{attribute 'GeneratedUsingTerminal: EK1122-0000-0018'}
{attribute addProperty BoxType "EK1122-0000-0018"}
{attribute addProperty Id "RP30_VI_AES_D_BC_ECAT_xAES_A3B0707168RP30_SAFETY_Flexi_Soft_EtherCAT_GatewayFlexi_Soft_EtherCAT_Gateway_DE394EDD5RP30_AB0_EPP1322_0001EPP1322_1FC0878B2RP30_AB1_EPP1008_0001EPP1008_78E8D3DD12RP30_AB2_EPP1008_0001EPP1008_78E8D3DD12RP30_AB3_EPP1008_0001EPP1008_78E8D3DD12RP30_AB4_EPP1008_0001EPP1008_78E8D3DD12"}
{attribute addProperty CRC "3284966580"}
{attribute addProperty Size "123"}
{attribute addProperty Name "RP30_A2 (EK1122)"}
TYPE RP30_A2_EK1122_C3CC9CB4 EXTENDS EK1122_1FC0878B :
STRUCT
    {attribute addProperty Name "RP30-VI (AES-D-BC-ECAT)"}
    {attribute addProperty PreviousPort "RP30_A2 (EK1122) : D"}
    {attribute addProperty SyncUnit "P30"}
    RP30_VI_AES_D_BC_ECAT_x : AES_A3B07071;
    {attribute addProperty Name "RP30-SAFETY (Flexi Soft EtherCAT Gateway)"}
    {attribute addProperty PreviousPort "RP30_A2 (EK1122) : B"}
    {attribute addProperty SyncUnit "P30"}
    RP30_SAFETY_Flexi_Soft_EtherCAT_Gateway : Flexi_Soft_EtherCAT_Gateway_DE394EDD;
    {attribute addProperty Name "RP30-AB0 (EPP1322-0001)"}
    {attribute addProperty PreviousPort "RP30-SAFETY (Flexi Soft EtherCAT Gateway) : B"}
    {attribute addProperty SyncUnit "default"}
    RP30_AB0_EPP1322_0001 : EPP1322_1FC0878B;
    {attribute addProperty Name "RP30-AB1 (EPP1008-0001)"}
    {attribute addProperty PreviousPort "RP30-AB0 (EPP1322-0001) : C"}
    {attribute addProperty SyncUnit "P30"}
    RP30_AB1_EPP1008_0001 : EPP1008_78E8D3DD;
    {attribute addProperty Name "RP30-AB2 (EPP1008-0001)"}
    {attribute addProperty PreviousPort "RP30-AB1 (EPP1008-0001) : B"}
    {attribute addProperty SyncUnit "P30"}
    RP30_AB2_EPP1008_0001 : EPP1008_78E8D3DD;
    {attribute addProperty Name "RP30-AB3 (EPP1008-0001)"}
    {attribute addProperty PreviousPort "RP30-AB2 (EPP1008-0001) : B"}
    {attribute addProperty SyncUnit "P30"}
    RP30_AB3_EPP1008_0001 : EPP1008_78E8D3DD;
    {attribute addProperty Name "RP30-AB4 (EPP1008-0001)"}
    {attribute addProperty PreviousPort "RP30-AB3 (EPP1008-0001) : B"}
    {attribute addProperty SyncUnit "P30"}
    RP30_AB4_EPP1008_0001 : EPP1008_78E8D3DD;
END_STRUCT
END_TYPE

(* stored: Version 1.2.0.0, ProductVersion 3.1.4024.11
   DUT RP30_A2_EK1122_C3CC9CB4: Id {cdc8526f-f695-0a3c-3af9-e89b6ce33bbe} *)
